// OptionalCyclic Plc -> Rob
AxesGroup.Config.PlcToRob.Header.TelegramNumberPlcToRob.00 := AxesGroup.Parameter.OptionalCyclic.PlcToRob.UseCallSubprogram;
AxesGroup.Config.PlcToRob.Header.TelegramNumberPlcToRob.01 := AxesGroup.Parameter.OptionalCyclic.PlcToRob.UseCartesianPos;
AxesGroup.Config.PlcToRob.Header.TelegramNumberPlcToRob.02 := AxesGroup.Parameter.OptionalCyclic.PlcToRob.UseJointPos;
AxesGroup.Config.PlcToRob.Header.TelegramNumberPlcToRob.03 := AxesGroup.Parameter.OptionalCyclic.PlcToRob.UseForce;
AxesGroup.Config.PlcToRob.Header.TelegramNumberPlcToRob.04 := AxesGroup.Parameter.OptionalCyclic.PlcToRob.Bit04;
AxesGroup.Config.PlcToRob.Header.TelegramNumberPlcToRob.05 := AxesGroup.Parameter.OptionalCyclic.PlcToRob.Bit05;
AxesGroup.Config.PlcToRob.Header.TelegramNumberPlcToRob.06 := AxesGroup.Parameter.OptionalCyclic.PlcToRob.Bit06;
AxesGroup.Config.PlcToRob.Header.TelegramNumberPlcToRob.07 := AxesGroup.Parameter.OptionalCyclic.PlcToRob.Bit07;  
AxesGroup.Config.PlcToRob.Header.TelegramNumberPlcToRob.08 := AxesGroup.Parameter.OptionalCyclic.PlcToRob.UseTwoSequences;
AxesGroup.Config.PlcToRob.Header.TelegramNumberPlcToRob.09 := AxesGroup.Parameter.OptionalCyclic.PlcToRob.UseCartesianPositionExt;
AxesGroup.Config.PlcToRob.Header.TelegramNumberPlcToRob.10 := AxesGroup.Parameter.OptionalCyclic.PlcToRob.UseJointPositionExt;
AxesGroup.Config.PlcToRob.Header.TelegramNumberPlcToRob.11 := AxesGroup.Parameter.OptionalCyclic.PlcToRob.Bit11;
AxesGroup.Config.PlcToRob.Header.TelegramNumberPlcToRob.12 := AxesGroup.Parameter.OptionalCyclic.PlcToRob.Bit12;
AxesGroup.Config.PlcToRob.Header.TelegramNumberPlcToRob.13 := AxesGroup.Parameter.OptionalCyclic.PlcToRob.Bit13;
AxesGroup.Config.PlcToRob.Header.TelegramNumberPlcToRob.14 := AxesGroup.Parameter.OptionalCyclic.PlcToRob.Bit14;
AxesGroup.Config.PlcToRob.Header.TelegramNumberPlcToRob.15 := AxesGroup.Parameter.OptionalCyclic.PlcToRob.Bit15;  

// OptionalCyclic Rob -> Plc
AxesGroup.Config.PlcToRob.Header.TelegramNumberPlcToRob.00 := AxesGroup.Parameter.OptionalCyclic.RobToPlc.UseCallSubprogram;
AxesGroup.Config.PlcToRob.Header.TelegramNumberPlcToRob.01 := AxesGroup.Parameter.OptionalCyclic.RobToPlc.UseCartesianPos;
AxesGroup.Config.PlcToRob.Header.TelegramNumberPlcToRob.02 := AxesGroup.Parameter.OptionalCyclic.RobToPlc.UseJointPos;
AxesGroup.Config.PlcToRob.Header.TelegramNumberPlcToRob.03 := AxesGroup.Parameter.OptionalCyclic.RobToPlc.UseForce;
AxesGroup.Config.PlcToRob.Header.TelegramNumberPlcToRob.04 := AxesGroup.Parameter.OptionalCyclic.RobToPlc.UseCurrent;
AxesGroup.Config.PlcToRob.Header.TelegramNumberPlcToRob.05 := AxesGroup.Parameter.OptionalCyclic.RobToPlc.Bit05;
AxesGroup.Config.PlcToRob.Header.TelegramNumberPlcToRob.06 := AxesGroup.Parameter.OptionalCyclic.RobToPlc.Bit06;
AxesGroup.Config.PlcToRob.Header.TelegramNumberPlcToRob.07 := AxesGroup.Parameter.OptionalCyclic.RobToPlc.Bit07;  
AxesGroup.Config.PlcToRob.Header.TelegramNumberPlcToRob.08 := AxesGroup.Parameter.OptionalCyclic.RobToPlc.UseTwoSequences;
AxesGroup.Config.PlcToRob.Header.TelegramNumberPlcToRob.09 := AxesGroup.Parameter.OptionalCyclic.RobToPlc.UseCartesianPositionExt;
AxesGroup.Config.PlcToRob.Header.TelegramNumberPlcToRob.10 := AxesGroup.Parameter.OptionalCyclic.RobToPlc.UseJointPositionExt;
AxesGroup.Config.PlcToRob.Header.TelegramNumberPlcToRob.11 := AxesGroup.Parameter.OptionalCyclic.RobToPlc.UseForceExt;
AxesGroup.Config.PlcToRob.Header.TelegramNumberPlcToRob.12 := AxesGroup.Parameter.OptionalCyclic.RobToPlc.UseCurrentEct;
AxesGroup.Config.PlcToRob.Header.TelegramNumberPlcToRob.13 := AxesGroup.Parameter.OptionalCyclic.RobToPlc.Bit13;  
AxesGroup.Config.PlcToRob.Header.TelegramNumberPlcToRob.14 := AxesGroup.Parameter.OptionalCyclic.RobToPlc.Bit14;
AxesGroup.Config.PlcToRob.Header.TelegramNumberPlcToRob.15 := AxesGroup.Parameter.OptionalCyclic.RobToPlc.Bit15;  


AxesGroup.Config.PlcToRob.Header.ClientDate := DATE_TO_IEC_DATE(DATE#2024-06-01 ); {warning 'ToDo: Get current date from target system'}
AxesGroup.Config.PlcToRob.Header.ClientTime := TIME_TO_IEC_TIME(TOD#12:00:00.000); {warning 'ToDo: Get current time from target system'}

// reset all variables
SendData.Reset();

// PlcToRob.Cyclic {{{
  
// PlcToRob.Cyclic.SRCIVersion  
SendData.AddByte     (VersionToByte(AxesGroup.Config.PlcToRob.Header.SRCIVersion));
// PlcToRob.Cyclic.FastStop_LifeSign
SendData.AddHalfBytes(AxesGroup.Config.PlcToRob.Header.FastStop, AxesGroup.Config.PlcToRob.Header.LifeSign); 
// PlcToRob.Cyclic.TelegramLengthPlcToRob
SendData.AddUint     (AxesGroup.Config.PlcToRob.Header.TelegramLengthPlcToRob);
// PlcToRob.Cyclic.TelegramLengthRobToPlc 
SendData.AddUint     (AxesGroup.Config.PlcToRob.Header.TelegramLengthRobToPlc);
// PlcToRob.Cyclic.AxesGroupID_Control
SendData.AddHalfBytes(AxesGroup.Config.PlcToRob.Header.AxesGroupID, AxesGroup.Config.PlcToRob.Header.Control);
// PlcToRob.Cyclic.Reserved
SendData.AddByte     (AxesGroup.Config.PlcToRob.Header.Reserved);
// PlcToRob.Cyclic.TelegramNumberPlcToRob 
SendData.AddUint     (AxesGroup.Config.PlcToRob.Header.TelegramNumberPlcToRob);
// PlcToRob.Cyclic.TelegramNumberRobToPlc 
SendData.AddUint     (AxesGroup.Config.PlcToRob.Header.TelegramNumberRobToPlc);
// PlcToRob.Cyclic.ClientDate
SendData.AddUint     (AxesGroup.Config.PlcToRob.Header.ClientDate); 
// PlcToRob.Cyclic.ClientTime
SendData.AddTime     (AxesGroup.Config.PlcToRob.Header.ClientTime);  
// }}}

// PlcToRob.CyclicOptional Data {{{

// AxesGroup.OptionalCyclic.PlcToRob.SubProgramData {{{
IF ( AxesGroup.OptionalCyclic.PlcToRob.SubProgramData.Active )
THEN
  SendData.AddDataBlock( ADR(AxesGroup.OptionalCyclic.PlcToRob.SubProgramData.Data), SIZEOF(AxesGroup.OptionalCyclic.PlcToRob.SubProgramData.Data));  
END_IF
// }}}

// AxesGroup.OptionalCyclic.PlcToRob.CartesianPos {{{
IF ( AxesGroup.OptionalCyclic.PlcToRob.CartesianPosition.Active) 
THEN
  // AxesGroup.OptionalCyclic.PlcToRob.CartesianPos.X
  SendData.AddReal(AxesGroup.OptionalCyclic.PlcToRob.CartesianPosition.X);
  // AxesGroup.OptionalCyclic.PlcToRob.CartesianPos.Y
  SendData.AddReal( AxesGroup.OptionalCyclic.PlcToRob.CartesianPosition.Y);
  // AxesGroup.OptionalCyclic.PlcToRob.CartesianPos.Z
  SendData.AddReal( AxesGroup.OptionalCyclic.PlcToRob.CartesianPosition.Z);
  // AxesGroup.OptionalCyclic.PlcToRob.CartesianPos.Rx
  SendData.AddReal( AxesGroup.OptionalCyclic.PlcToRob.CartesianPosition.Rx);
  // AxesGroup.OptionalCyclic.PlcToRob.CartesianPos.Ry
  SendData.AddReal( AxesGroup.OptionalCyclic.PlcToRob.CartesianPosition.Ry);
  // AxesGroup.OptionalCyclic.PlcToRob.CartesianPos.Rz
  SendData.AddReal( AxesGroup.OptionalCyclic.PlcToRob.CartesianPosition.Rz);
  // AxesGroup.OptionalCyclic.PlcToRob.CartesianPos.Config
 _tmpByte   := 0;
 _tmpByte.0 := AxesGroup.OptionalCyclic.PlcToRob.CartesianPosition.Config.Shoulder = ArmConfigShoulder.BACK;
 _tmpByte.1 := AxesGroup.OptionalCyclic.PlcToRob.CartesianPosition.Config.Elbow    = ArmConfigElbow   .DOWN;
 _tmpByte.2 := AxesGroup.OptionalCyclic.PlcToRob.CartesianPosition.Config.Wrist    = ArmConfigWrist   .FLIP;
 
  SendData.AddByte(_tmpByte);
          
  // AxesGroup.OptionalCyclic.PlcToRob.CartesianPos.TurnNumber.J1 + J2
  SendData.AddHalfBytes( SINT_TO_BYTE(AxesGroup.OptionalCyclic.PlcToRob.CartesianPosition.TurnNumber.J1Turns), SINT_TO_BYTE(AxesGroup.OptionalCyclic.PlcToRob.CartesianPosition.TurnNumber.J2Turns));
  // AxesGroup.OptionalCyclic.PlcToRob.CartesianPos.TurnNumber.J3 + J4
  SendData.AddHalfBytes( SINT_TO_BYTE(AxesGroup.OptionalCyclic.PlcToRob.CartesianPosition.TurnNumber.J3Turns), SINT_TO_BYTE(AxesGroup.OptionalCyclic.PlcToRob.CartesianPosition.TurnNumber.J4Turns));
  // AxesGroup.OptionalCyclic.PlcToRob.CartesianPos.TurnNumber.J5 + J6
  SendData.AddHalfBytes( SINT_TO_BYTE(AxesGroup.OptionalCyclic.PlcToRob.CartesianPosition.TurnNumber.J5Turns), SINT_TO_BYTE(AxesGroup.OptionalCyclic.PlcToRob.CartesianPosition.TurnNumber.J6Turns));
  // AxesGroup.OptionalCyclic.PlcToRob.CartesianPos.TurnNumber.E1 
  SendData.AddSint(AxesGroup.OptionalCyclic.PlcToRob.CartesianPosition.TurnNumber.E1Turns);
  // AxesGroup.OptionalCyclic.PlcToRob.CartesianPos.E1
  SendData.AddReal( AxesGroup.OptionalCyclic.PlcToRob.CartesianPosition.E1);
  // AxesGroup.OptionalCyclic.PlcToRob.CartesianPos.CoordinateSystem.ToolNo
  SendData.AddUsint(AxesGroup.OptionalCyclic.PlcToRob.CartesianPosition.CoordinateSystem.ToolNo);
  // AxesGroup.OptionalCyclic.PlcToRob.CartesianPos.CoordinateSystem.FrameNo 
  SendData.AddUsint(AxesGroup.OptionalCyclic.PlcToRob.CartesianPosition.CoordinateSystem.FrameNo);  
END_IF
// }}}
  
// AxesGroup.OptionalCyclic.PlcToRob.CartesianPosExt {{{
IF ( AxesGroup.OptionalCyclic.PlcToRob.CartesianPositionExt.Active) 
THEN
  // AxesGroup.OptionalCyclic.PlcToRob.CartesianPosExt.E2 
  SendData.AddReal( AxesGroup.OptionalCyclic.PlcToRob.CartesianPositionExt.E2);
  // AxesGroup.OptionalCyclic.PlcToRob.CartesianPosExt.E3
  SendData.AddReal( AxesGroup.OptionalCyclic.PlcToRob.CartesianPositionExt.E3);
  // AxesGroup.OptionalCyclic.PlcToRob.CartesianPosExt.E4
  SendData.AddReal( AxesGroup.OptionalCyclic.PlcToRob.CartesianPositionExt.E4);
  // AxesGroup.OptionalCyclic.PlcToRob.CartesianPosExt.E5
  SendData.AddReal( AxesGroup.OptionalCyclic.PlcToRob.CartesianPositionExt.E5);
  // AxesGroup.OptionalCyclic.PlcToRob.CartesianPosExt.E6
  SendData.AddReal( AxesGroup.OptionalCyclic.PlcToRob.CartesianPositionExt.E6);
END_IF    
// }}}
      
// AxesGroup.OptionalCyclic.PlcToRob.JointPosition {{{
IF ( AxesGroup.OptionalCyclic.PlcToRob.JointPosition.Active) 
THEN
  // AxesGroup.OptionalCyclic.PlcToRob.JointPosition.J1
  SendData.AddReal( AxesGroup.OptionalCyclic.PlcToRob.JointPosition.J1);
  // AxesGroup.OptionalCyclic.PlcToRob.JointPosition.J2
  SendData.AddReal( AxesGroup.OptionalCyclic.PlcToRob.JointPosition.J2);
  // AxesGroup.OptionalCyclic.PlcToRob.JointPosition.J3
  SendData.AddReal( AxesGroup.OptionalCyclic.PlcToRob.JointPosition.J3);
  // AxesGroup.OptionalCyclic.PlcToRob.JointPosition.J4
  SendData.AddReal( AxesGroup.OptionalCyclic.PlcToRob.JointPosition.J4);
  // AxesGroup.OptionalCyclic.PlcToRob.JointPosition.J5
  SendData.AddReal( AxesGroup.OptionalCyclic.PlcToRob.JointPosition.J5);
  // AxesGroup.OptionalCyclic.PlcToRob.JointPosition.J6
  SendData.AddReal( AxesGroup.OptionalCyclic.PlcToRob.JointPosition.J6);
  // AxesGroup.OptionalCyclic.PlcToRob.JointPosition.E1
  SendData.AddReal( AxesGroup.OptionalCyclic.PlcToRob.JointPosition.E1);
END_IF
// }}}

// AxesGroup.OptionalCyclic.PlcToRob.JointPositionExt {{{
IF ( AxesGroup.OptionalCyclic.PlcToRob.JointPositionExt.Active) 
THEN
  // AxesGroup.OptionalCyclic.PlcToRob.JointPositionExt.E2
  SendData.AddReal( AxesGroup.OptionalCyclic.PlcToRob.JointPositionExt.E2);
  // AxesGroup.OptionalCyclic.PlcToRob.JointPositionExt.E3
  SendData.AddReal( AxesGroup.OptionalCyclic.PlcToRob.JointPositionExt.E3);  
  // AxesGroup.OptionalCyclic.PlcToRob.JointPositionExt.E4
  SendData.AddReal( AxesGroup.OptionalCyclic.PlcToRob.JointPositionExt.E4);
  // AxesGroup.OptionalCyclic.PlcToRob.JointPositionExt.E5
  SendData.AddReal( AxesGroup.OptionalCyclic.PlcToRob.JointPositionExt.E5);
  // AxesGroup.OptionalCyclic.PlcToRob.JointPositionExt.E6
  SendData.AddReal( AxesGroup.OptionalCyclic.PlcToRob.JointPositionExt.E6);        
END_IF  
// }}}
     
// AxesGroup.OptionalCyclic.PlcToRob.CartesianForce {{{
IF ( AxesGroup.OptionalCyclic.PlcToRob.CartesianForce.Active) 
THEN
  // AxesGroup.OptionalCyclic.PlcToRob.CartesianForce.X
  SendData.AddReal( AxesGroup.OptionalCyclic.PlcToRob.CartesianForce.X);
  // AxesGroup.OptionalCyclic.PlcToRob.CartesianForce.Y
  SendData.AddReal( AxesGroup.OptionalCyclic.PlcToRob.CartesianForce.Y);
  // AxesGroup.OptionalCyclic.PlcToRob.CartesianForce.Z
  SendData.AddReal( AxesGroup.OptionalCyclic.PlcToRob.CartesianForce.Z);
  // AxesGroup.OptionalCyclic.PlcToRob.CartesianForce.Rx
  SendData.AddReal( AxesGroup.OptionalCyclic.PlcToRob.CartesianForce.Rx);
  // AxesGroup.OptionalCyclic.PlcToRob.CartesianForce.Ry
  SendData.AddReal( AxesGroup.OptionalCyclic.PlcToRob.CartesianForce.Ry);
  // AxesGroup.OptionalCyclic.PlcToRob.CartesianForce.Rz
  SendData.AddReal( AxesGroup.OptionalCyclic.PlcToRob.CartesianForce.Rz);
END_IF  
// }}}
                    
// AxesGroup.OptionalCyclic.PlcToRob.CartesianForceExt {{{
IF ( AxesGroup.OptionalCyclic.PlcToRob.CartesianForceExt.Active) 
THEN
  // AxesGroup.OptionalCyclic.PlcToRob.CartesianForceExt.E1
  SendData.AddReal( AxesGroup.OptionalCyclic.PlcToRob.CartesianForceExt.E1);
  // AxesGroup.OptionalCyclic.PlcToRob.CartesianForceExt.E2
  SendData.AddReal( AxesGroup.OptionalCyclic.PlcToRob.CartesianForceExt.E2);
  // AxesGroup.OptionalCyclic.PlcToRob.CartesianForceExt.E3
  SendData.AddReal( AxesGroup.OptionalCyclic.PlcToRob.CartesianForceExt.E3);
  // AxesGroup.OptionalCyclic.PlcToRob.CartesianForceExt.E4
  SendData.AddReal( AxesGroup.OptionalCyclic.PlcToRob.CartesianForceExt.E4);
  // AxesGroup.OptionalCyclic.PlcToRob.CartesianForceExt.E5
  SendData.AddReal( AxesGroup.OptionalCyclic.PlcToRob.CartesianForceExt.E5);
  // AxesGroup.OptionalCyclic.PlcToRob.CartesianForceExt.E6
  SendData.AddReal( AxesGroup.OptionalCyclic.PlcToRob.CartesianForceExt.E6);
END_IF                    


// }}}

// }}}
  
{warning 'ToDo: Sequence Handling for Seq 0..1'}
// PlcToRob.Sequence[0]{{{

// PlcToRob.Sequence[0].Header{{{
  
// AxesGroup.OptionalCyclic.PlcToRob.Sequence[0].Header.SEQ_ACK 
SendData.AddUint( Telegram.PlcToRob.Sequence[0].Header.SEQ_ACK);
// AxesGroup.OptionalCyclic.PlcToRob.Sequence[0].Header.PayloadLength
SendData.AddUint( Telegram.PlcToRob.Sequence[0].Header.PayloadLength);
// }}}

    
{warning 'ToDo: Fragment Handling for Frag 0..9'}
// PlcToRob.Sequence[0].Fragment {{{

       
          
// PlcToRob.Sequence[0].Fragment.Header {{{

// AxesGroup.OptionalCyclic.PlcToRob.Sequence[0].Fragment.Header.ID 
SendData.AddUint( Telegram.PlcToRob.Sequence[0].Fragment[0].Header.ID);
// AxesGroup.OptionalCyclic.PlcToRob.Sequence[0].Fragment.Header.Reserve
SendData.AddByte(Telegram.PlcToRob.Sequence[0].Fragment[0].Header.Reserve);
// AxesGroup.OptionalCyclic.PlcToRob.Sequence[0].Fragment.Header.FragmentAction 
SendData.AddByte(FragmentActionToByte(Telegram.PlcToRob.Sequence[0].Fragment[0].Header.FragmentAction));
// AxesGroup.OptionalCyclic.PlcToRob.Sequence[0].Fragment.Header.PayloadPointer
SendData.AddUint(Telegram.PlcToRob.Sequence[0].Fragment[0].Header.PayloadPointer);
// AxesGroup.OptionalCyclic.PlcToRob.Sequence[0].Fragment.Header.PayloadLength 
SendData.AddUint(Telegram.PlcToRob.Sequence[0].Fragment[0].Header.PayloadLength);

// PlcToRob.Sequence[0].Fragment.Command {{{    
FOR _payLoadPtr := AxesGroup.Acyclic.ActiveCommandRegister.Register[1].Command[1].PayLoadPtr TO AxesGroup.Acyclic.ActiveCommandRegister.Register[1].Command[1].PayloadLen   
DO
  // copy payload
  SendData.AddByte(AxesGroup.Acyclic.ActiveCommandRegister.Register[1].Command[1].Payload[_payLoadPtr]);

  // inc payload pointer
  AxesGroup.Acyclic.ActiveCommandRegister.Register[1].Command[1].PayLoadPtr 
    := AxesGroup.Acyclic.ActiveCommandRegister.Register[1].Command[1].PayLoadPtr + 1;

  // set command state
  IF ( AxesGroup.Acyclic.ActiveCommandRegister.Register[1].Command[1].PayLoadPtr >= AxesGroup.Acyclic.ActiveCommandRegister.Register[1].Command[1].PayLoadLen) 
  THEN
    AxesGroup.Acyclic.ActiveCommandRegister.Register[1].Command[1].State := BufferStateCmd.PROCESSED;
  ELSE
    AxesGroup.Acyclic.ActiveCommandRegister.Register[1].Command[1].State := BufferStateCmd.SENDING;  
  END_IF 

  // check limit reached ?
  IF ( SendData.PayloadLen >= RobotLibraryParameter.ROBOT_OUT_DATA_MAX - SIZEOF(Telegram.PlcToRob.Footer)) 
  THEN
    EXIT;
  END_IF  
END_FOR    
// }}}
// }}}
// }}}
// }}}


// Footer {{{

// PlcToRob.Footer.Reserved_LifeSign
SendData.AddHalfBytes(0, AxesGroup.Config.PlcToRob.Header.LifeSign);

// }}}

                      
END_METHOD

METHOD NetworkLayer
VAR_IN_OUT
  /// Robot assignment of function
  AxesGroup         : AxesGroup;
    /// Inputs of PLC for communication from RC
  RobotInData       : ARRAY[1..RobotLibraryParameter.ROBOT_IN_DATA_MAX ] OF BYTE;
  /// Outputs of PLC for communication to RC
  RobotOutData      : ARRAY[1..RobotLibraryParameter.ROBOT_OUT_DATA_MAX] OF BYTE;
END_VAR
                        CreateSendData   ( AxesGroup    := AxesGroup,
                   RobotInData  := RobotInData,
                   RobotOutData := RobotOutData );

ParseRecvData    ( AxesGroup    := AxesGroup,
                   RobotInData  := RobotInData,
                   RobotOutData := RobotOutData );                   
                      
END_METHOD

METHOD OnCall
VAR_IN_OUT
   /// Robot assignment of function
  AxesGroup : AxesGroup;
END_VAR
                        
                      
END_METHOD

METHOD ParseRecvData
VAR_IN_OUT
  /// Robot assignment of function
  AxesGroup    : AxesGroup;
  /// Inputs of PLC for communication from RC
  RobotInData  : ARRAY[1..RobotLibraryParameter.ROBOT_IN_DATA_MAX ] OF BYTE;
  /// Outputs of PLC for communication to RC
  RobotOutData : ARRAY[1..RobotLibraryParameter.ROBOT_OUT_DATA_MAX] OF BYTE;
END_VAR

VAR
  /// internal index
 _idx             : DINT;
  /// temporary DWORD
 _tmpDword        : DWORD;
  /// length of data block
 _dataBlockLength : UINT;
  /// internal payload length
 _payLoadLen      : DWORD;  
  /// internal payload pointer
 _payLoadPtr      : DWORD;  
END_VAR
                        // Version
AxesGroup.Config.RobToPlc.Header.SRCIVersion.MajorVersion := RecvData.GetUsint();
AxesGroup.Config.RobToPlc.Header.SRCIVersion.MinorVersion := RecvData.GetUsint();
AxesGroup.Config.RobToPlc.Header.SRCIVersion.PatchVersion := RecvData.GetUsint();
// Connection alive signal
AxesGroup.Config.RobToPlc.Header.LifeSign       := RecvData.GetByte();
// Reserved byte
AxesGroup.Config.RobToPlc.Header.Reserved       := RecvData.GetByte();
// Initialization and Telegram control state
AxesGroup.Config.RobToPlc.Header.TelegramState  := RecvData.GetUsint();
// Combination of various RA related states.
AxesGroup.Config.RobToPlc.Header.StatusRobotArm := DwordToRaStatusWord(RecvData.GetDword());
// Actual override in percentage encoding 
AxesGroup.Config.RobToPlc.Header.Override       := RecvData.GetUint();


// AxesGroup.OptionalCyclic {{{

// AxesGroup.OptionalCyclic.RobToPlc.SubProgramData {{{
IF ( AxesGroup.OptionalCyclic.RobToPlc.SubProgramData.Active )
THEN
  FOR _idx := 0 TO 25 DO
    AxesGroup.Config.RobToPlc.CyclicOptional.SubProgramData.Data[_idx] := RecvData.GetByte(); 
	END_FOR
END_IF
// }}}
  
// AxesGroup.OptionalCyclic.RobToPlc.CartesianPos {{{
IF ( AxesGroup.OptionalCyclic.RobToPlc.CartesianPosition.Active )
THEN
  AxesGroup.Config.RobToPlc.CyclicOptional.CartesianPosition.X                    := RecvData.GetReal();
  AxesGroup.Config.RobToPlc.CyclicOptional.CartesianPosition.Y                    := RecvData.GetReal();
  AxesGroup.Config.RobToPlc.CyclicOptional.CartesianPosition.Z                    := RecvData.GetReal();
  AxesGroup.Config.RobToPlc.CyclicOptional.CartesianPosition.Rx                   := RecvData.GetReal();
  AxesGroup.Config.RobToPlc.CyclicOptional.CartesianPosition.Ry                   := RecvData.GetReal();
  AxesGroup.Config.RobToPlc.CyclicOptional.CartesianPosition.Rz                   := RecvData.GetReal();
  AxesGroup.Config.RobToPlc.CyclicOptional.CartesianPosition.Config               := RecvData.GetArmConfig();
  AxesGroup.Config.RobToPlc.CyclicOptional.CartesianPosition.TurnNumber           := RecvData.GetTurnNumbers();
  AxesGroup.Config.RobToPlc.CyclicOptional.CartesianPosition.E1                   := RecvData.GetReal();  
  AxesGroup.Config.RobToPlc.CyclicOptional.CartesianPosition.E2                   := RecvData.GetReal();
  AxesGroup.Config.RobToPlc.CyclicOptional.CartesianPosition.E3                   := RecvData.GetReal();
  AxesGroup.Config.RobToPlc.CyclicOptional.CartesianPosition.E4                   := RecvData.GetReal();
  AxesGroup.Config.RobToPlc.CyclicOptional.CartesianPosition.E5                   := RecvData.GetReal();
  AxesGroup.Config.RobToPlc.CyclicOptional.CartesianPosition.E6                   := RecvData.GetReal();      
  AxesGroup.Config.RobToPlc.CyclicOptional.CartesianPosition.ToolNo               := RecvData.GetUsint();
  AxesGroup.Config.RobToPlc.CyclicOptional.CartesianPosition.FrameNo              := RecvData.GetUsint();
  AxesGroup.Config.RobToPlc.CyclicOptional.CartesianPosition.CurrentlyUsedToolNo  := RecvData.GetUsint();
  AxesGroup.Config.RobToPlc.CyclicOptional.CartesianPosition.CurrentlyUsedFrameNo := RecvData.GetUsint();
  AxesGroup.Config.RobToPlc.CyclicOptional.CartesianPosition.Reserve_1            := RecvData.GetByte();
  AxesGroup.Config.RobToPlc.CyclicOptional.CartesianPosition.Reserve_2            := RecvData.GetByte();  
END_IF
// }}}

// AxesGroup.OptionalCyclic.RobToPlc.CartesianPosExt {{{
IF ( AxesGroup.OptionalCyclic.RobToPlc.CartesianPositionExt.Active )
THEN
  AxesGroup.Config.RobToPlc.CyclicOptional.CartesianPositionExt.E2 := RecvData.GetReal();
  AxesGroup.Config.RobToPlc.CyclicOptional.CartesianPositionExt.E3 := RecvData.GetReal();
  AxesGroup.Config.RobToPlc.CyclicOptional.CartesianPositionExt.E4 := RecvData.GetReal();
  AxesGroup.Config.RobToPlc.CyclicOptional.CartesianPositionExt.E5 := RecvData.GetReal();
  AxesGroup.Config.RobToPlc.CyclicOptional.CartesianPositionExt.E6 := RecvData.GetReal();
END_IF  
// }}}       

// AxesGroup.OptionalCyclic.RobToPlc.JointPosition {{{
IF ( AxesGroup.OptionalCyclic.RobToPlc.JointPosition.Active )
THEN
  AxesGroup.Config.RobToPlc.CyclicOptional.JointPosition.J1         := RecvData.GetReal();
  AxesGroup.Config.RobToPlc.CyclicOptional.JointPosition.J2         := RecvData.GetReal();
  AxesGroup.Config.RobToPlc.CyclicOptional.JointPosition.J3         := RecvData.GetReal();
  AxesGroup.Config.RobToPlc.CyclicOptional.JointPosition.J4         := RecvData.GetReal();
  AxesGroup.Config.RobToPlc.CyclicOptional.JointPosition.J5         := RecvData.GetReal();
  AxesGroup.Config.RobToPlc.CyclicOptional.JointPosition.J6         := RecvData.GetReal();
  AxesGroup.Config.RobToPlc.CyclicOptional.JointPosition.E1         := RecvData.GetReal();
  AxesGroup.Config.RobToPlc.CyclicOptional.JointPosition.E1_Reserve := RecvData.GetWord();
END_IF  
// }}}
  
// AxesGroup.OptionalCyclic.RobToPlc.JointPosition {{{
IF ( AxesGroup.OptionalCyclic.RobToPlc.JointPositionExt.Active )
THEN
  AxesGroup.Config.RobToPlc.CyclicOptional.JointPositionExt.E2 := RecvData.GetReal();
  AxesGroup.Config.RobToPlc.CyclicOptional.JointPositionExt.E3 := RecvData.GetReal();
  AxesGroup.Config.RobToPlc.CyclicOptional.JointPositionExt.E4 := RecvData.GetReal();
  AxesGroup.Config.RobToPlc.CyclicOptional.JointPositionExt.E5 := RecvData.GetReal();
  AxesGroup.Config.RobToPlc.CyclicOptional.JointPositionExt.E6 := RecvData.GetReal();  
END_IF  
// }}}    
      
// AxesGroup.OptionalCyclic.RobToPlc.CartesianForce {{{
IF ( AxesGroup.OptionalCyclic.RobToPlc.CartesianForce.Active )
THEN
  AxesGroup.Config.RobToPlc.CyclicOptional.Force.X  := RecvData.GetReal();
  AxesGroup.Config.RobToPlc.CyclicOptional.Force.Y  := RecvData.GetReal();
  AxesGroup.Config.RobToPlc.CyclicOptional.Force.Z  := RecvData.GetReal();
  AxesGroup.Config.RobToPlc.CyclicOptional.Force.Rx := RecvData.GetReal();
  AxesGroup.Config.RobToPlc.CyclicOptional.Force.Ry := RecvData.GetReal();
  AxesGroup.Config.RobToPlc.CyclicOptional.Force.Rz := RecvData.GetReal();
END_IF  
// }}}    
      
// AxesGroup.OptionalCyclic.RobToPlc.CartesianForceExt {{{
IF ( AxesGroup.OptionalCyclic.RobToPlc.CartesianForceExt.Active )
THEN
  AxesGroup.Config.RobToPlc.CyclicOptional.ForceExt.E1  := RecvData.GetReal();
  AxesGroup.Config.RobToPlc.CyclicOptional.ForceExt.E2  := RecvData.GetReal();
  AxesGroup.Config.RobToPlc.CyclicOptional.ForceExt.E3  := RecvData.GetReal();
  AxesGroup.Config.RobToPlc.CyclicOptional.ForceExt.E4  := RecvData.GetReal();
  AxesGroup.Config.RobToPlc.CyclicOptional.ForceExt.E5  := RecvData.GetReal();
  AxesGroup.Config.RobToPlc.CyclicOptional.ForceExt.E6  := RecvData.GetReal();
END_IF
// }}}    

// AxesGroup.OptionalCyclic.RobToPlc.Current {{{
IF ( AxesGroup.OptionalCyclic.RobToPlc.JointCurrent.Active )
THEN
  AxesGroup.Config.RobToPlc.CyclicOptional.Current.J1  := RecvData.GetReal();
  AxesGroup.Config.RobToPlc.CyclicOptional.Current.J2  := RecvData.GetReal();
  AxesGroup.Config.RobToPlc.CyclicOptional.Current.J3  := RecvData.GetReal();
  AxesGroup.Config.RobToPlc.CyclicOptional.Current.J4  := RecvData.GetReal();
  AxesGroup.Config.RobToPlc.CyclicOptional.Current.J5  := RecvData.GetReal();
  AxesGroup.Config.RobToPlc.CyclicOptional.Current.J6  := RecvData.GetReal();
END_IF
// }}}    
  
// AxesGroup.OptionalCyclic.RobToPlc.CurrentExt {{{
IF ( AxesGroup.OptionalCyclic.RobToPlc.JointCurrentExt.Active )
THEN
  AxesGroup.Config.RobToPlc.CyclicOptional.CurrentExt.E1  := RecvData.GetReal();
  AxesGroup.Config.RobToPlc.CyclicOptional.CurrentExt.E2  := RecvData.GetReal();
  AxesGroup.Config.RobToPlc.CyclicOptional.CurrentExt.E3  := RecvData.GetReal();
  AxesGroup.Config.RobToPlc.CyclicOptional.CurrentExt.E4  := RecvData.GetReal();
  AxesGroup.Config.RobToPlc.CyclicOptional.CurrentExt.E5  := RecvData.GetReal();
  AxesGroup.Config.RobToPlc.CyclicOptional.CurrentExt.E6  := RecvData.GetReal();
END_IF
// }}}
    
// }}}    

// Sequence Data
AxesGroup.Config.RobToPlc.Sequence[0].Header.SEQ_ACK       := RecvData.GetUint();
AxesGroup.Config.RobToPlc.Sequence[0].Header.PayloadLength := RecvData.GetUint();

AxesGroup.Config.RobToPlc.Sequence[0].Fragment[1].Header.ID                  := RecvData.GetUint();
AxesGroup.Config.RobToPlc.Sequence[0].Fragment[1].Header.Reserve             := RecvData.GetByte();
AxesGroup.Config.RobToPlc.Sequence[0].Fragment[1].Header.FragmentAction      := RecvData.GetFragmentAction();
AxesGroup.Config.RobToPlc.Sequence[0].Fragment[1].Header.PayloadPointer      := RecvData.GetUint();
AxesGroup.Config.RobToPlc.Sequence[0].Fragment[1].Header.PayloadLength       := RecvData.GetUint();

AxesGroup.Config.RobToPlc.Sequence[0].Fragment[1].Command.Header.CmdType     := RecvData.GetUint();
AxesGroup.Config.RobToPlc.Sequence[0].Fragment[1].Command.Header.Prio        := RecvData.GetByte();
AxesGroup.Config.RobToPlc.Sequence[0].Fragment[1].Command.Header.ExecMode    := RecvData.GetUsint();
AxesGroup.Config.RobToPlc.Sequence[0].Fragment[1].Command.Header.ParSequence := RecvData.GetByte();


_dataBlockLength :=           AxesGroup.Config.RobToPlc.Sequence[0].Fragment[1].Header.PayloadLength 
                    -  SIZEOF(AxesGroup.Config.RobToPlc.Sequence[0].Fragment[1].Command.Header); 

FOR _idx := 1 TO  _dataBlockLength
DO
  AxesGroup.Config.RobToPlc.Sequence[0].Fragment[1].Command.Payload[_idx] := RecvData.GetByte();
END_FOR

WHILE (RecvData.PayloadPtr < 1)
DO
;  
END_WHILE
                      
END_METHOD

METHOD TransportLayer
VAR_IN_OUT
   /// Robot assignment of function
  AxesGroup : AxesGroup;
END_VAR
                        
                      
END_METHOD
END_FUNCTION_BLOCK

/// Calculate frame with three-point method
FUNCTION_BLOCK CalculateFrameFB EXTENDS RobotLibraryBaseFB
// ------------------------------------------------------------------------- 
//  SRCI Robot Library                                                
// ------------------------------------------------------------------------- 
//                                                                           
//  Object:      CalculateFrameFB                                       
//  Author:      Thorsten Brach                                                
//  Date:        2024-06-01
//
//  Description:                                              
//   
//                                                                           
//  Copyright: 
//    (C) 2024 Thorsten Brach. All rights reserved                                                                         
//                                                                           
//  Disclaimer:                                                                           
//    This project is provided without any guarantee and can be used for   
//    private and commercial purposes. Any commercial use is at the user’s 
//    own risk and responsibility.
//
// -------------------------------------------------------------------------
VAR_INPUT
  /// Start of the command at the rising edge
  Execute            : BOOL;
  /// Define which method should be used to calculate the tool frame
  Mode               : FrameCalculationMode;
  /// Index of target frame
  /// • 0: WCS (default)
  /// • 1..254: User frames
  FrameNo            : USINT;  
  /// Cartesian position in the positive direction of the  X-Axis of the calculated frame coordinate system relative to the given frame
  Position_X         : RobotCartesianPosition;
  /// Cartesian position in the XY-plane of the calculated frame coordinate system relative to the given frame.
  Position_XY        : RobotCartesianPosition;
  /// Cartesian position of the origin of the calculated frame coordinate system relative to the given frame.
  Position_Origin    : RobotCartesianPosition;
  /// Cartesian position of the postponement of the origin of the calculated frame coordinate system relative to the given frame.
  /// Auxiliary position if the origin of the can’t be reached by the robot, i.e. because it is inside an object.
  OriginShift        : RobotCartesianPosition;
  /// Index of frame on which the calculated frame is depending
  /// •      0: WCS (default)
  /// • 1..254: User frames
  ReferenceFrame     : USINT;
END_VAR
VAR_OUTPUT
  /// The command has been completed successfully
  Done               : BOOL;
  /// FB is being processed
  Busy               : BOOL;
  /// Command is transferred and confirmed by the RC
  CommandBuffered    : BOOL;
  /// Frame data
  FrameData           : FrameData;
END_VAR

                  
                

METHOD PROTECTED OnCall
VAR_IN_OUT
  /// Robot assignment of function
  AxesGroup         : AxesGroup; 
END_VAR
                        
                      
END_METHOD
END_FUNCTION_BLOCK

/// Calculate Inverse Kinematic
FUNCTION_BLOCK CalculateInverseKinematicFB EXTENDS RobotLibraryBaseFB
// ------------------------------------------------------------------------- 
//  SRCI Robot Library                                                
// ------------------------------------------------------------------------- 
//                                                                           
//  Object:      CalculateInverseKinematicFB                                       
//  Author:      Thorsten Brach                                                
//  Date:        2024-06-01
//
//  Description:                                              
//   
//                                                                           
//  Copyright: 
//    (C) 2024 Thorsten Brach. All rights reserved                                                                         
//                                                                           
//  Disclaimer:                                                                           
//    This project is provided without any guarantee and can be used for   
//    private and commercial purposes. Any commercial use is at the user’s 
//    own risk and responsibility.
//
// -------------------------------------------------------------------------
VAR_INPUT
  /// Start of the command at the rising edge
  Execute            : BOOL;
  /// cartesian position
  CartesianPosition  : RobotCartesianPosition;
  /// Index of target tool
  /// • 0: Flange (default)
  /// • 1..254: Tool frames
  ToolNo             : USINT;
  /// Index of target frame
  /// • 0: WCS (default)
  /// • 1..254: User frames
  FrameNo            : USINT;  
END_VAR
VAR_OUTPUT
  /// The command has been completed successfully
  Done               : BOOL;
  /// FB is being processed
  Busy               : BOOL;
  /// Command is transferred and confirmed by the RC
  CommandBuffered    : BOOL;
  /// Calculated robot joint position
  JointPosition      : RobotJointPosition;
END_VAR

                  
                

METHOD PROTECTED OnCall
VAR_IN_OUT
  /// Robot assignment of function
  AxesGroup         : AxesGroup; 
END_VAR
                        
                      
END_METHOD
END_FUNCTION_BLOCK

/// Calculate tool (TCP) with four-point method
FUNCTION_BLOCK CalculateToolFB EXTENDS RobotLibraryBaseFB
// ------------------------------------------------------------------------- 
//  SRCI Robot Library                                                
// ------------------------------------------------------------------------- 
//                                                                           
//  Object:      CalculateToolFB                                       
//  Author:      Thorsten Brach                                                
//  Date:        2024-06-01
//
//  Description:                                              
//   
//                                                                           
//  Copyright: 
//    (C) 2024 Thorsten Brach. All rights reserved                                                                         
//                                                                           
//  Disclaimer:                                                                           
//    This project is provided without any guarantee and can be used for   
//    private and commercial purposes. Any commercial use is at the user’s 
//    own risk and responsibility.
//
// -------------------------------------------------------------------------
VAR_INPUT
  /// Start of the command at the rising edge
  Execute            : BOOL;
  /// Define which method should be used to calculate the tool frame
  Mode               : ToolCalculationMode;
  /// Index of target tool
  /// • 0: Flange (default)
  /// • 1..254: Tool frames
  ToolNo             : USINT;
  /// Index of target frame
  /// • 0: WCS (default)
  /// • 1..254: User frames
  FrameNo            : USINT;  
  /// • True: Tool fixed
  /// • False: Tool on flange (default)
  ExternalTCP        : BOOL;
  /// Positions in cartesian coordinates for the tool frame calculation.
  PositionsArray     : ARRAY[0..5] OF RobotCartesianPosition;
END_VAR
VAR_OUTPUT
  /// The command has been completed successfully
  Done               : BOOL;
  /// FB is being processed
  Busy               : BOOL;
  /// Command is transferred and confirmed by the RC
  CommandBuffered    : BOOL;
  /// Tool data
  ToolData           : ToolData;
  /// Maximum error of deviation of the TCP position
  /// from the fix point in world coordinate system
  /// If not supported: • -1
  TCPMaxError       : REAL;
  /// Average error of TCP position from the fix point  in world coordinate system
  /// If not supported: • -1 
  TCPMeanError      : REAL;
END_VAR

                  
                

METHOD PROTECTED OnCall
VAR_IN_OUT
  /// Robot assignment of function
  AxesGroup         : AxesGroup; 
END_VAR
                        
                      
END_METHOD
END_FUNCTION_BLOCK

/// Activate conveyor tracking mode
FUNCTION_BLOCK ActivateConveyorTrackingFB EXTENDS RobotLibraryBaseFB
// ------------------------------------------------------------------------- 
//  SRCI Robot Library                                                
// ------------------------------------------------------------------------- 
//                                                                           
//  Object:      ActivateConveyorTrackingFB                                       
//  Author:      Thorsten Brach                                                
//  Date:        2024-06-01
//
//  Description:                                              
//   
//                                                                           
//  Copyright: 
//    (C) 2024 Thorsten Brach. All rights reserved                                                                         
//                                                                           
//  Disclaimer:                                                                           
//    This project is provided without any guarantee and can be used for   
//    private and commercial purposes. Any commercial use is at the user’s 
//    own risk and responsibility.
//
// -------------------------------------------------------------------------
VAR_INPUT
  /// Set TRUE to change RA power state to "Enabled"
  Enable             : BOOL;
  /// Index of assigned conveyor
  ConveyorNo         : USINT;
  /// Specifies encoder connection setup (at least one option must be supported)
  ConnectionMode     : ConnectionMode;
  /// Relates to "ConnectionMode" 1 – "PLC connected": Value of the encoder connected to the conveyor belt
  PLCEncoderValue    : REAL;
END_VAR

VAR_OUTPUT
  /// TRUE, while the following outputs return valid values:
  /// • TrackingStatusByte
  /// • RCEncoderValue
  Valid              : BOOL;
  /// FB is being processed
  Busy               : BOOL;
  /// Command is transferred and confirmed by the RC
  CommandBuffered    : BOOL;
  /// Receiving of input parameter values has been acknowledged by RC
  ParameterAccepted  : BOOL;
  /// Current status of "ConveyorTracking" according to Table 6-432
  TrackingStatus     : TrackingStatus;
  /// Relates to "ConnectionMode" 1 – "RC connected": Traveled distance of assigned conveyor since ConveyorTracking has been activated (offset)
  RCEncoderValue     : REAL;
END_VAR

                  
                

METHOD Protected OnCall
VAR_IN_OUT
  /// Robot assignment of function
  AxesGroup         : AxesGroup; 
END_VAR
                        
                      
END_METHOD
END_FUNCTION_BLOCK

/// Configure conveyor parameters
FUNCTION_BLOCK ConfigureConveyorFB EXTENDS RobotLibraryBaseFB
// ------------------------------------------------------------------------- 
//  SRCI Robot Library                                                
// ------------------------------------------------------------------------- 
//                                                                           
//  Object:      ConfigureConveyorFB                                       
//  Author:      Thorsten Brach                                                
//  Date:        2024-06-01
//
//  Description:                                              
//   
//                                                                           
//  Copyright: 
//    (C) 2024 Thorsten Brach. All rights reserved                                                                         
//                                                                           
//  Disclaimer:                                                                           
//    This project is provided without any guarantee and can be used for   
//    private and commercial purposes. Any commercial use is at the user’s 
//    own risk and responsibility.
//
// -------------------------------------------------------------------------
VAR_INPUT
  /// Start of the command at the rising edge
  Execute            : BOOL;
  /// Index of assigned conveyor
  ConveyorNo         : USINT;  
  ///Define the origin coordinate system of the conveyor belt, with the X-Axis pointing in the direction of the movement of the conveyor belt.
  ConveyorOrigin     : FrameData;
  /// Define the type of the conveyor
  ConveyorType       : ConveyorType;
  /// Relates to "ConveyorType" "Circular Tracking": Define the radius of the circular conveyor
  Radius             : REAL;
  /// Distance [mm] from the origin of the conveyor belt to the beginning of the "SyncInZone"
  StartDistance      : REAL;
  /// Distance [mm] from the origin of the conveyor belt to the end of the "SyncOutZone"
  EndDistance        : REAL;
  /// Define the length of the "SyncInZone"
  SyncInLength       : REAL;
  /// Define the length of the "SyncOutZone"
  SyncOutLength      : REAL;
END_VAR

VAR_OUTPUT
  /// The command has been completed successfully
  Done               : BOOL;
  /// FB is being processed
  Busy               : BOOL;
  /// Command is transferred and confirmed by the RC
  CommandBuffered    : BOOL;
END_VAR

                  
                

METHOD PROTECTED OnCall
VAR_IN_OUT
  /// Robot assignment of function
  AxesGroup         : AxesGroup; 
END_VAR
                        
                      
END_METHOD
END_FUNCTION_BLOCK

/// Redefine tracking position for conveyor tracking
FUNCTION_BLOCK RedefineTrackingPosFB EXTENDS RobotLibraryBaseFB
// ------------------------------------------------------------------------- 
//  SRCI Robot Library                                                
// ------------------------------------------------------------------------- 
//                                                                           
//  Object:      RedefineTrackingPosFB                                       
//  Author:      Thorsten Brach                                                
//  Date:        2024-06-01
//
//  Description:                                              
//   
//                                                                           
//  Copyright: 
//    (C) 2024 Thorsten Brach. All rights reserved                                                                         
//                                                                           
//  Disclaimer:                                                                           
//    This project is provided without any guarantee and can be used for   
//    private and commercial purposes. Any commercial use is at the user’s 
//    own risk and responsibility.
//
// -------------------------------------------------------------------------
VAR_INPUT
  /// Start of the command at the rising edge
  Execute                : BOOL;
  /// Relates to ListenerID >0:
  ProcessingMode         : ProcessingMode;
  /// Index of assigned conveyor
  ConveyorNo             : USINT;
  /// Relates to ListenerID = 0:
  /// Define initial work piece position relative to the conveyor belt origin:
  /// • Origin (X, Y, Z in mm)
  /// • Orientation (RX, RY, RZ in degree)
  /// For more information refer to chapter 5.5.14.
  InitObjectPosition     : ARRAY[0..5] OF REAL;
  /// Relates to ListenerID = 0:
  /// Travel distance of assigned UCS between work piece detection (InitObjectPosition) and execution of this command.
  TrackingOffset         : REAL;
  /// Relates to ListenerID >0
  /// Start index of real registers containing InitObjectPosition for trigger-based execution.
  StartIndexInitPosition : INT;
  /// Define the index number of the UCS that is assigned to the conveyor by the function "ConveyorTracking".
  /// For more information refer to chapter 5.5.14.
  FrameNo                : USINT;
  /// Relates to ListenerID >0
  /// Index of real register containing TrackingOffset for trigger-based execution
  IndexTrackingOffset    : USINT;
  /// ID of associated trigger function:
  /// • 0: No Trigger (default): No trigger related behavior
  /// • >0: Trigger: o Start executing, when the trigger function with the identical EmitterID is triggered.
  /// Always positive.
  /// For more information, see chapter 5.5.12 Triggers
  ListenerID             :  SINT;
END_VAR

VAR_OUTPUT
  /// The command has been completed successfully
  Done                   : BOOL;
  /// FB is being processed
  Busy                   : BOOL;
  /// Command is transferred and confirmed by the RC
  CommandBuffered        : BOOL;
  /// Receiving of input parameter values has been acknowledged by RC
  ParameterAccepted      : BOOL;
  /// Unique system-generated ID of the "Action" when the function is triggered.
  /// • >0: The "Action" is started by the trigger funcrion with identical FollowID.
  /// • <0: The "Action" is stopped by the trigger function with identical FollowID.
  /// For more information see chapter 5.5.12.4 EmitterID, ListenerID, FollowID and OriginID
  OriginID               : INT;
  /// Relates to ListenerID >0
  /// Number of successful trigger-based command invocations - For more information refer TO chapter 5.5.12.4
  InvocationCounter      : USINT;
END_VAR

                  
                

METHOD PROTECTED OnCall
VAR_IN_OUT
  /// Robot assignment of function
  AxesGroup         : AxesGroup; 
END_VAR
                        
                      
END_METHOD
END_FUNCTION_BLOCK

/// Synchronize robot with conveyor
FUNCTION_BLOCK SyncToConveyorFB EXTENDS RobotLibraryBaseFB
// ------------------------------------------------------------------------- 
//  SRCI Robot Library                                                
// ------------------------------------------------------------------------- 
//                                                                           
//  Object:      SyncToConveyorFB                                       
//  Author:      Thorsten Brach                                                
//  Date:        2024-06-01
//
//  Description:                                              
//   
//                                                                           
//  Copyright: 
//    (C) 2024 Thorsten Brach. All rights reserved                                                                         
//                                                                           
//  Disclaimer:                                                                           
//    This project is provided without any guarantee and can be used for   
//    private and commercial purposes. Any commercial use is at the user’s 
//    own risk and responsibility.
//
// -------------------------------------------------------------------------
VAR_INPUT
  /// Start of the command at the rising edge
  Execute            : BOOL;
  /// Index of assigned conveyor
  ConveyorNo         : USINT;
  /// Define the index number of the UCS that will be assigned to the conveyor.
  /// For more information refer to chapter 5.5.14
  FrameNo            : USINT;
  /// Defines when synchronization starts
  SyncInMode         : SyncInMode;
  /// Relates to "SyncInMode" "After distance" (1) and "After time" (2): Parameter for the synchronization
  /// • "After distance" (1) -  Distance in mm
  /// • "After time" (2) -  Time in ms
  SyncInParameter    : REAL;
  /// Define the maximum adjustment velocity for the robot to catch up to the conveyor belt.
  /// The velocity must be greater than the velocity of the conveyor belt.
  /// • 0 (default): no limit - No conveyor tracking specific limit
  ///                         - RC internal limit applies
  /// • >0: use limit         - Conveyor tracking specific limit applies
  MaxVelocity        : REAL;
  /// Define the maximum adjustment acceleration for the robot to catch up to the conveyor belt.
  /// • 0 (default): no limit - No conveyor tracking specific limit
  ///                         - RC internal limit applies
  /// • >0: use limit         - Conveyor tracking specific limit applies
  MaxAcceleration    : REAL;
  /// ID of associated trigger function:
  /// • 0: No Trigger (default): No trigger related behavior
  /// • >0: Trigger:  Start executing, when the trigger function with the identical EmitterID is triggered.
  /// Always positive.
  /// For more information, see chapter 5.5.12 Triggers
  ListenerID         : SINT;
END_VAR

VAR_OUTPUT
  /// FB is being processed
  Busy               : BOOL;
  /// Command is transferred and confirmed by the RC
  CommandBuffered    : BOOL;
  /// TRUE, while SyncToConveyor is enabled and processing input parameters
  Enabled            : BOOL;
  /// The command takes control of the motion of the according axis group
  Active             : BOOL;
  /// The command was aborted by another command.
  CommandAborted     : BOOL;
  /// Receiving of input parameter values has been acknowledged by RC
  ParameterAccepted  : BOOL;
  /// The TCP is in synchronization with the object on the conveyor belt.
  InSync             : BOOL;
  /// Unique system-generated ID of the "Action" when the function is triggered.
  /// • >0: The "Action" is started by the trigger function with identical FollowID.
  /// • <0: The "Action" is stopped by the trigger function with identical FollowID.
  /// For more information see chapter 5.5.12.4 EmitterID, ListenerID, FollowID and OriginID
  OriginID           : INT;
  /// Relates to ListenerID >0
  /// Number of successful trigger -based command invocations
  /// For more information refer to chapter 5.5.12.4.
  InvocationCounter  : USINT;
END_VAR

                  
                

METHOD PROTECTED OnCall
VAR_IN_OUT
  /// Robot assignment of function
  AxesGroup         : AxesGroup; 
END_VAR
                        
                      
END_METHOD
END_FUNCTION_BLOCK

/// Enables the RC to apply user defined force/ torque through RA’s TCP movement
FUNCTION_BLOCK ForceControlFB EXTENDS RobotLibraryBaseFB
// ------------------------------------------------------------------------- 
//  SRCI Robot Library                                                
// ------------------------------------------------------------------------- 
//                                                                           
//  Object:      ForceControlFB                                       
//  Author:      Thorsten Brach                                                
//  Date:        2024-06-01
//
//  Description:                                              
//   
//                                                                           
//  Copyright: 
//    (C) 2024 Thorsten Brach. All rights reserved                                                                         
//                                                                           
//  Disclaimer:                                                                           
//    This project is provided without any guarantee and can be used for   
//    private and commercial purposes. Any commercial use is at the user’s 
//    own risk and responsibility.
//
// -------------------------------------------------------------------------
VAR_INPUT
  /// Start of the command at the rising edge
  Execute            : BOOL;
  /// Defines type of reference of Force and Torque (at least one option must be supported)
  ReferenceType      : ReferenceType;
  /// Relates to ConnectionMode 1 and 2 (Sensor connected to PLC).
  /// Currently applied force and torque detected by sensor according to ReferenceType, ToolNo and FrameNo.
  /// • [0]: X-Axis
  /// • [1]: Y-Axis
  /// • [2]: Z- Axis
  /// • [3]: Rotation around X-Axis (RX)
  /// • [4]: Rotation around Y-Axis (RY)
  /// • [5]: Rotation around Z- Axis (RZ)
  SensorValue        : ARRAY[0..5] OF REAL;
  /// Relates to ReferenceType 0 (Tool) and 1 (Frame):
  /// Force and torque to be applied by robot arm according to ReferenceType, ToolNo and FrameNo:
  /// • [0]: X-Axis
  /// • [1]: Y-Axis
  /// • [2]: Z- Axis
  /// • [3]: Rotation around X-Axis (RX)
  /// • [4]: Rotation around Y-Axis (RY)
  /// • [5]: Rotation around Z- Axis (RZ)
  /// Set TargetValue <>-99999.9999 (default) to define setpoint
  TargetValue        : ARRAY[0..5] OF REAL;
  /// Index of tool
  /// •      0: Flange (default)
  /// • 1..254: Tool frames
  ToolNo             : USINT;
  /// Define the index number of the UCS that will be assigned to the conveyor.
  /// For more information refer to chapter 5.5.14
  FrameNo            : USINT;
  /// Specifies encoder connection setup according to Table 6-713 (at least one option must be supported) 
  ConnectionMode     : SensorConnectionMode;
  /// Position of sensor relative to flange (FixedSensor FALSE) or relative to WCS (FixedSensor TRUE)
  /// • [0]: X-Axis
  /// • [1]: Y-Axis
  /// • [2]: Z- Axis
  /// • [3]: Rotation around X-Axis (RX)
  /// • [4]: Rotation around Y-Axis (RY)
  /// • [5]: Rotation around Z- Axis (RZ)
  SensorFrame        : ARRAY[0..5] OF REAL;
  /// Index of payload data containing mass, center of gravity, orientation and inertia relative to SensorFrame.
  /// Required to calibrate system for setting up gravity compensation and sensor offset.
  CalibrationData    : USINT;
  /// Tolerance of TargetValue within which currently applied force/torque will return ForceStatus "Specified force/torque reached" TRUE.
  TargetWindow       : REAL;
  /// Define axes whose position may be adjusted by the robot to apply specified force according to Table 6-711.
  CompliantAxes      : BYTE;
  /// Maximum allowed TCP velocity for compliant axes in % of nominal velocity.
  /// •   0% (default): no limit - RC internal limit applies
  /// •  >0% use limit -  Specified limit applies
  /// • 100% use maximal reference velocity
  /// For more information on nominal dynamics see chapter 5.5.7 Robot dynamics 
  MaxVelocity        : REAL;
  /// Maximum allowed cartesian deviation according to ReferenceType, ToolNo and FrameNo.
  /// Set 0 (default) to not specify a limit in this axis direction.
  /// • [0]: Deviation in X-Direction in mm
  /// • [1]: Deviation in Y- direction in mm
  /// • [2]: Deviation in Z- direction in mm
  /// • [3]: Deviation in RX- direction in °
  /// • [4]: Deviation in RY- direction in °
  /// • [5]: Deviation in RZ- direction in °
  MaxDeviation       : ARRAY [0..5] OF REAL;
  /// Defines reaction in case ForceControl reports error during its execution
  /// Processing of active move command is continued without active ForceControl
  ErrorReaction      : ErrorReaction;
  /// Relates to ErrorReaction 0 (Abort and move). Defines type of reference coordinate system of ErrorVector
  ErrorReferenceType : ReferenceType;
  /// Relates to ErrorReaction 0 (Abort and move). Vector defining robot’s movement in case of
  /// incoming error according to ErrorReferenceType, ErrorToolNo and ErrorFrameNo.
  /// • [0]: X-Axis
  /// • [1]: Y-Axis
  /// • [2]: Z- Axis
  /// • [3]: Rotation around X-Axis (RX)
  /// • [4]: Rotation around Y-Axis (RY)
  /// • [5]: Rotation around Z-Axis (RZ)
  ErrorVector        : ARRAY [0..5] OF REAL;
  /// Relates to ErrorReaction 0 (Abort and move). Index of tool.
  /// • 0 (default): Flange
  /// • 1..254: Tool frames
  ErrorToolNo        : USINT;
  /// Relates to ErrorReferenceType 1 (Frame)
  /// •      0: WCS (default)
  /// • 1..254: User frames
  ErrorFrameNo       : USINT;
  /// Defines sensor positioning:
  /// • FALSE (default): Sensor mounted on flange
  /// • TRUE: Sensor fixed
  FixedSensor        : BOOL;
END_VAR

VAR_OUTPUT
  /// TRUE, while the following outputs return valid values:
  /// - ForceStatus
  Valid              : BOOL;
  /// FB is being processed
  Busy               : BOOL;
  /// Command is transferred and confirmed by the RC
  CommandBuffered    : BOOL;
  /// Receiving of input parameter values has been acknowledged by RC
  ParameterAccepted  : BOOL;
  /// Current status of ForceControl and ForceLimit (chapter 6.5.25) according to Table 6-712
  ForceStatus        : ForceStatus;
END_VAR

                  
                

METHOD PROTECTED OnCall
VAR_IN_OUT
  /// Robot assignment of function
  AxesGroup         : AxesGroup; 
END_VAR
                        
                      
END_METHOD
END_FUNCTION_BLOCK

/// Commands specified reaction from RA when defined force/torque detected
FUNCTION_BLOCK ForceLimitFB EXTENDS RobotLibraryBaseFB
// ------------------------------------------------------------------------- 
//  SRCI Robot Library                                                
// ------------------------------------------------------------------------- 
//                                                                           
//  Object:      ForceLimitFB                                       
//  Author:      Thorsten Brach                                                
//  Date:        2024-06-01
//
//  Description:                                              
//   
//                                                                           
//  Copyright: 
//    (C) 2024 Thorsten Brach. All rights reserved                                                                         
//                                                                           
//  Disclaimer:                                                                           
//    This project is provided without any guarantee and can be used for   
//    private and commercial purposes. Any commercial use is at the user’s 
//    own risk and responsibility.
//
// -------------------------------------------------------------------------
VAR_INPUT
  /// Start of the command at the rising edge
  Execute            : BOOL;
  /// Defines type of reference of Force and Torque (at least one option must be supported)
  ReferenceType      : ReferenceType;
  /// Relates to ConnectionMode 1 and 2 (Sensor connected to PLC).
  /// Currently applied force and torque detected by sensor according to ReferenceType, ToolNo and FrameNo.
  /// • [0]: X-Axis
  /// • [1]: Y-Axis
  /// • [2]: Z- Axis
  /// • [3]: Rotation around X-Axis (RX)
  /// • [4]: Rotation around Y-Axis (RY)
  /// • [5]: Rotation around Z- Axis (RZ)
  SensorValue        : ARRAY[0..5] OF REAL;
  /// Index of tool
  /// •      0: Flange (default)
  /// • 1..254: Tool frames
  ToolNo             : USINT;
  /// Define the index number of the UCS that will be assigned to the conveyor.
  /// For more information refer to chapter 5.5.14
  FrameNo            : USINT;
  /// Maximal allowed force and torque detected by the sensor according to ReferenceType and ToolNo/FrameNo before robot reacts according to ReactionMode.
  /// Set value <>0 (default) to monitor coordinate axes
  /// • [0]: X-Axis
  /// • [1]: Y-Axis
  /// • [2]: Z- Axis
  /// • [3]: Rotation around X-Axis (RX)
  /// • [4]: Rotation around Y-Axis (RY)
  /// • [5]: Rotation around Z- Axis (RZ)
  ForceLimit        : ARRAY[0..5] OF REAL;
  /// Specifies encoder connection setup according to Table 6-713 (at least one option must be supported) 
  ConnectionMode    : SensorConnectionMode;
  /// Position of sensor relative to flange (FixedSensor FALSE) or relative to WCS (FixedSensor TRUE)
  /// • [0]: X-Axis
  /// • [1]: Y-Axis
  /// • [2]: Z- Axis
  /// • [3]: Rotation around X-Axis (RX)
  /// • [4]: Rotation around Y-Axis (RY)
  /// • [5]: Rotation around Z- Axis (RZ)
  SensorFrame        : ARRAY[0..5] OF REAL;
  /// Index of payload data containing mass, center of gravity, orientation and inertia relative to SensorFrame.
  /// Required to calibrate system for setting up gravity compensation and sensor offset.
  CalibrationData    : USINT;
  /// Defines sensor positioning:
  /// • FALSE (default): Sensor mounted on flange
  /// • TRUE: Sensor fixed
  FixedSensor        : BOOL;
  /// ID of Action that will be executed when this command is active
  /// • >0: Start Action        - Start executing the Action function with the identical ListenerID.
  /// • <0: Stop Action         - Stop executing the Action function with the identical ListenerID.
  /// •  0: Undefined (default) - If no EmitterID is defined, the function returns an error message
  /// For more information see chapter 5.5.12.4
  EmitterID          : SINT;  
END_VAR

VAR_OUTPUT
  /// TRUE, while the following outputs return valid values
  Valid              : BOOL;
  /// FB is being processed
  Busy               : BOOL;
  /// Command is transferred and confirmed by the RC
  CommandBuffered    : BOOL;
  /// Receiving of input parameter values has been acknowledged by RC
  ParameterAccepted  : BOOL;
  /// Current status of ForceControl and ForceLimit (chapter 6.5.25) according to Table 6-712
  ForceStatus        : ForceStatus;
  /// Relates to EmitterID <> 0: Unique system-generated ID of the trigger function when the function is called by user.
  /// For more information see chapter 5.5.12.4.
  FollowID           : DINT;
END_VAR

                  
                

METHOD PROTECTED OnCall
VAR_IN_OUT
  /// Robot assignment of function
  AxesGroup         : AxesGroup; 
END_VAR
                        
                      
END_METHOD
END_FUNCTION_BLOCK

/// Read actual force/torque at TCP
FUNCTION_BLOCK ReadActualForceFB EXTENDS RobotLibraryBaseFB
// ------------------------------------------------------------------------- 
//  SRCI Robot Library                                                
// ------------------------------------------------------------------------- 
//                                                                           
//  Object:      ReadActualForceFB                                       
//  Author:      Thorsten Brach                                                
//  Date:        2024-06-01
//
//  Description:                                              
//   
//                                                                           
//  Copyright: 
//    (C) 2024 Thorsten Brach. All rights reserved                                                                         
//                                                                           
//  Disclaimer:                                                                           
//    This project is provided without any guarantee and can be used for   
//    private and commercial purposes. Any commercial use is at the user’s 
//    own risk and responsibility.
//
// -------------------------------------------------------------------------
VAR_INPUT
  /// Start of the command at the rising edge
  Execute            : BOOL;
  /// Processing Mode
  ProcessingMode      : ProcessingMode;
  /// Defines type of reference of Force and Torque (at least one option must be supported )
  ReferenceType       : ReferenceType;
  /// Index of tool
  /// •      0: Flange (default)
  /// • 1..254: Tool frames
  ToolNo             : USINT;
  /// Define the index number of the UCS that will be assigned to the conveyor.
  /// For more information refer to chapter 5.5.14
  FrameNo            : USINT;
  /// Index of payload data containing mass, center of gravity, orientation and inertia relative to SensorFrame.
  /// Required to calibrate system for setting up gravity compensation and sensor offset.
  CalibrationData    : USINT;
  /// ID of associated trigger function:
  /// • 0: Immediately (default) - Start executing this function immediately.
  /// • >0: Trigger -  Start executing, when the trigger function with the identical EmitterID is triggered.
  /// Always positive.
  /// For more information, see chapter 5.5.12 Triggers
  ListenerID         : SINT;
 
END_VAR

VAR_OUTPUT
  /// TRUE, when command has been completed successfully.
  Done               : BOOL;
  /// TRUE, while the following outputs return valid values:
  /// - ActualForce
  Valid              : BOOL;
  /// FB is being processed
  Busy               : BOOL;
  /// Command is transferred and confirmed by the RC
  CommandBuffered    : BOOL;
  /// Receiving of input parameter values has been acknowledged by RC
  ParameterAccepted  : BOOL;
  /// Currently detected force and torque according to ReferenceType, ToolNo and FrameNo.
  /// • [0]: X-Axis
  /// • [1]: Y-Axis
  /// • [2]: Z- Axis
  /// • [3]: Rotation around X-Axis (RX)
  /// • [4]: Rotation around Y-Axis (RY)
  /// • [5]: Rotation around Z- Axis (RZ)
  ActualForce        : ARRAY[0..5] OF REAL;
  /// Unique system-generated ID of the "Action" when the function is triggered.
  /// • >0: The "Action" is started by the trigger function with identical FollowID.
  /// • <0: The "Action" is stopped by the trigger function with identical FollowID.
  /// For more information see chapter 5.5.12.4 EmitterID, ListenerID, FollowID and OriginID
  OriginID           : INT;
  /// Relates to ListenerID >0
  /// Number of successful trigger -based command invocations
  /// For more information refer to chapter 5.5.12.4.
  InvocationCounter  : USINT;
  
END_VAR

                  
                

METHOD PROTECTED OnCall
VAR_IN_OUT
  /// Robot assignment of function
  AxesGroup         : AxesGroup; 
END_VAR
                        
                      
END_METHOD
END_FUNCTION_BLOCK

/// Continue interrupted path
FUNCTION_BLOCK GroupContinueFB EXTENDS RobotLibraryBaseFB
// ------------------------------------------------------------------------- 
//  SRCI Robot Library                                                
// ------------------------------------------------------------------------- 
//                                                                           
//  Object:      GroupContinueFB                                       
//  Author:      Thorsten Brach                                                
//  Date:        2024-06-01
//
//  Description:                                              
//   
//                                                                           
//  Copyright: 
//    (C) 2024 Thorsten Brach. All rights reserved                                                                         
//                                                                           
//  Disclaimer:                                                                           
//    This project is provided without any guarantee and can be used for   
//    private and commercial purposes. Any commercial use is at the user’s 
//    own risk and responsibility.
//
// -------------------------------------------------------------------------
VAR_INPUT
  /// Start of the command at the rising edge
  Execute            : BOOL;
END_VAR
VAR_OUTPUT
  /// The command has been completed successfully
  Done               : BOOL;
  /// FB is being processed
  Busy               : BOOL;
  /// Command is transferred and confirmed by the RC
  CommandBuffered    : BOOL;
END_VAR

                  
                

METHOD PROTECTED OnCall
VAR_IN_OUT
  /// Robot assignment of function
  AxesGroup         : AxesGroup; 
END_VAR
                        
                      
END_METHOD
END_FUNCTION_BLOCK

/// Interrupt active movement, possible to continue movement
FUNCTION_BLOCK GroupInterruptFB EXTENDS RobotLibraryBaseFB
// ------------------------------------------------------------------------- 
//  SRCI Robot Library                                                
// ------------------------------------------------------------------------- 
//                                                                           
//  Object:      GroupInterruptFB                                       
//  Author:      Thorsten Brach                                                
//  Date:        2024-06-01
//
//  Description:                                              
//   
//                                                                           
//  Copyright: 
//    (C) 2024 Thorsten Brach. All rights reserved                                                                         
//                                                                           
//  Disclaimer:                                                                           
//    This project is provided without any guarantee and can be used for   
//    private and commercial purposes. Any commercial use is at the user’s 
//    own risk and responsibility.
//
// -------------------------------------------------------------------------
VAR_INPUT
  /// Start of the command at the rising edge
  Execute            : BOOL;
END_VAR

VAR_OUTPUT
  /// The command has been completed successfully
  Done               : BOOL;
  /// FB is being processed
  Busy               : BOOL;
  /// Command is transferred and confirmed by the RC
  CommandBuffered    : BOOL;
  /// The command takes control of the motion of the according axis group.
  Active             : BOOL;
END_VAR

                  
                

METHOD PROTECTED OnCall
VAR_IN_OUT
  /// Robot assignment of function
  AxesGroup         : AxesGroup; 
END_VAR
                        
                      
END_METHOD
END_FUNCTION_BLOCK

/// Jog robot manually
FUNCTION_BLOCK GroupJogFB EXTENDS RobotLibraryBaseFB
// ------------------------------------------------------------------------- 
//  SRCI Robot Library                                                
// ------------------------------------------------------------------------- 
//                                                                           
//  Object:      GroupJogFB                                       
//  Author:      Thorsten Brach                                                
//  Date:        2024-06-01
//
//  Description:                                              
//   
//                                                                           
//  Copyright: 
//    (C) 2024 Thorsten Brach. All rights reserved                                                                         
//                                                                           
//  Disclaimer:                                                                           
//    This project is provided without any guarantee and can be used for   
//    private and commercial purposes. Any commercial use is at the user’s 
//    own risk and responsibility.
//
// -------------------------------------------------------------------------
VAR_INPUT
  /// Activate jog command
  Enable                 : BOOL;
  /// Specifies in which mode the robot is jogged
  Mode                   : JogMode;
  /// Velocity in % of monitoring speed or ReferenceVelocity, depending on the currently active operation mode 
  /// (T1 External/T2 External: Monitoring speed; Automatic External: ReferenceVelocity )
  /// •    0%: No movement of the robot
  /// •   10%: default
  /// • ≤100%: use input parameter value
  Override               : REAL;
  /// Change to jog and define direction according to Mode. See Table 6-223
  Control                : JogControl;
  /// Relates to Mode 0 (JogFrame) and 1 (JogTool) Index of tool
  /// •      0: Flange (default):
  /// • 1..254: Tool frames
  ToolNo                 : USINT;
  /// Relates to Mode 0 (JogFrame) Index of frame
  /// •      0: WCS (default)
  /// • 1..254: User frames
  FrameNo                : USINT;
  /// Increments for jogging translational axes for defined distance
  /// •  0: Incremental mode OFF (default) - Movement is active until "Control" is reset, or error occurs.
  /// • >0: Incremental mode ON            - Movement is active until distance defined by input value is reached without changes to "Control", "Control" is reset, or error occurs
  IncrementalTranslation : REAL;
  /// Increments for jogging rotational axes for defined distance
  /// • 0: Incremental mode OFF (default) - Movement is active until "Control" is reset, or error occurs.
  /// • >0 Incremental mode ON:           - Movement is active until distance defined by input value is reached without changes to "Control", "Control" is reset, or error occurs
  IncrementalRotation    : REAL;
END_VAR

VAR_OUTPUT
  /// Relates to Incremental mode ON: TRUE, when robot’s TCP or axes have traversed distance of "IncrementalTranslation" or "IncrementalRotation"
  DistanceReached        : BOOL;
  /// FB is being processed
  Busy                   : BOOL;
  /// Command is transferred and confirmed by the RC
  CommandBuffered        : BOOL;
  /// TRUE while GroupJog is enabled
  Enabled                : BOOL;
  /// The command takes control of the motion of the according axis group
  Active                 : BOOL;
  /// The active movement was aborted by another command
  CommandAborted         : BOOL;
  /// Receiving of input parameter values has been acknowledged by RC
  ParameterAccepted      : BOOL;
END_VAR

                  
                

METHOD PROTECTED OnCall
VAR_IN_OUT
  /// Robot assignment of function
  AxesGroup         : AxesGroup; 
END_VAR
                        
                      
END_METHOD
END_FUNCTION_BLOCK

/// Acknowledgement all pending errors
FUNCTION_BLOCK GroupResetFB EXTENDS RobotLibraryBaseFB
// ------------------------------------------------------------------------- 
//  SRCI Robot Library                                                
// ------------------------------------------------------------------------- 
//                                                                           
//  Object:      GroupResetFB                                       
//  Author:      Thorsten Brach                                                
//  Date:        2024-06-01
//
//  Description:                                              
//   
//                                                                           
//  Copyright: 
//    (C) 2024 Thorsten Brach. All rights reserved                                                                         
//                                                                           
//  Disclaimer:                                                                           
//    This project is provided without any guarantee and can be used for   
//    private and commercial purposes. Any commercial use is at the user’s 
//    own risk and responsibility.
//
// -------------------------------------------------------------------------
VAR_INPUT
  /// Start of the command at the rising edge
  Execute         : BOOL;
END_VAR

VAR_OUTPUT
  /// The command has been completed successfully
  Done            : BOOL;
  /// FB is being processed
  Busy            : BOOL;
  /// Command is transferred and confirmed by the RC
  CommandBuffered : BOOL;
END_VAR

                  
                

METHOD PROTECTED OnCall
VAR_IN_OUT
  /// Robot assignment of function
  AxesGroup         : AxesGroup; 
END_VAR
                        
                      
END_METHOD
END_FUNCTION_BLOCK

/// Abort actual movement and delete buffer
FUNCTION_BLOCK GroupStopFB EXTENDS RobotLibraryBaseFB
// ------------------------------------------------------------------------- 
//  SRCI Robot Library                                                
// ------------------------------------------------------------------------- 
//                                                                           
//  Object:      GroupStopFB                                       
//  Author:      Thorsten Brach                                                
//  Date:        2024-06-01
//
//  Description:                                              
//   
//                                                                           
//  Copyright: 
//    (C) 2024 Thorsten Brach. All rights reserved                                                                         
//                                                                           
//  Disclaimer:                                                                           
//    This project is provided without any guarantee and can be used for   
//    private and commercial purposes. Any commercial use is at the user’s 
//    own risk and responsibility.
//
// -------------------------------------------------------------------------
VAR_INPUT
  /// Start of the command at the rising edge
  Execute            : BOOL;
END_VAR

VAR_OUTPUT
  /// The command has been completed successfully
  Done               : BOOL;
  /// FB is being processed
  Busy               : BOOL;
  /// Command is transferred and confirmed by the RC
  CommandBuffered    : BOOL;
  /// Frame index
  AbortedSequence    : SequenceFlag;
END_VAR

                  
                

METHOD PROTECTED OnCall
VAR_IN_OUT
  /// Robot assignment of function
  AxesGroup         : AxesGroup; 
END_VAR
                        
                      
END_METHOD
END_FUNCTION_BLOCK

/// Automatic detection of load data
FUNCTION_BLOCK LoadMeasurementAutomaticFB EXTENDS RobotLibraryBaseFB
// ------------------------------------------------------------------------- 
//  SRCI Robot Library                                                
// ------------------------------------------------------------------------- 
//                                                                           
//  Object:      LoadMeasurementAutomaticFB                                       
//  Author:      Thorsten Brach                                                
//  Date:        2024-06-01
//
//  Description:                                              
//   
//                                                                           
//  Copyright: 
//    (C) 2024 Thorsten Brach. All rights reserved                                                                         
//                                                                           
//  Disclaimer:                                                                           
//    This project is provided without any guarantee and can be used for   
//    private and commercial purposes. Any commercial use is at the user’s 
//    own risk and responsibility.
//
// -------------------------------------------------------------------------
VAR_INPUT
  /// Start of the command at the rising edge
  Execute            : BOOL;
  /// Define which method should be used to measure the load data
  Mode               : LoadMeasurementMode;
  /// Parameter which determines the behavior towards the previously sent and still active or buffered commands.
  AbortingMode       : AbortingMode;
  /// Define which mass is expected as a result of the load measurement
  Mass               : REAL;
  /// Define the area for the allowed motion of the Joint 3. 
  /// The order of the two limit values does not matter. 
  /// Only considered with "Mode" = 0, 2.
  Area_J3            : ARRAY[0..1] OF REAL;
  /// Define the area for the allowed motion of the Joint 4. 
  /// The order of the two limit values does not matter. 
  /// Only considered with "Mode" = 0, 2.
  Area_J4            : ARRAY[0..1] OF REAL;
  /// Define the area for the allowed motion of the Joint 5. 
  /// The order of the two limit values does not matter. 
  /// Only considered with "Mode" = 0, 2.
  Area_J5            : ARRAY[0..1] OF REAL;
  /// Define the area for the allowed motion of the Joint 6. 
  /// The order of the two limit values does not matter. 
  /// Only considered with "Mode" = 0, 2.
  Area_J6            : ARRAY[0..1] OF REAL;
  /// Define the first position for the load measurement.
  /// Only considered with "Mode" = 0, 1.
  Position_1         : RobotJointPosition;
  /// Define the second position for the load measurement.
  /// Only considered with "Mode" = 3.
  Position_2         : RobotJointPosition;
  /// Define the configuration angle for the load measurement.
  /// Only considered with "Mode" = 1.
  ConfigurationAngle : REAL;
  /// Defines the target sequence in which the command will be executed
  SequenceFlag       : SequenceFlag;
END_VAR
VAR_OUTPUT
  ///The command has been completed successfully
  Done               : BOOL;
  /// FB is being processed
  Busy               : BOOL;
  /// Command is transferred and confirmed by the RC
  CommandBuffered    : BOOL;  
  /// The command takes control of the motion of the according axis group.
  Active             : BOOL;
  /// The command was aborted by another command.
  CommandAborted     : BOOL;
  /// TRUE, while command is interrupted during execution and can be continued.
  CommandInterrupted : BOOL;
  /// FB is returning a unique ID for the cal led measurement.
  MeasuringID        : UINT;
  /// Measured load data (see chapter 5.5.6.4)
  LoadData           : LoadData;
END_VAR

                  
                

METHOD PROTECTED OnCall
VAR_IN_OUT
  /// Robot assignment of function
  AxesGroup         : AxesGroup; 
END_VAR
                        
                      
END_METHOD
END_FUNCTION_BLOCK

/// Sequential detection of load data
FUNCTION_BLOCK LoadMeasurementSequentialFB EXTENDS RobotLibraryBaseFB
// ------------------------------------------------------------------------- 
//  SRCI Robot Library                                                
// ------------------------------------------------------------------------- 
//                                                                           
//  Object:      LoadMeasurementSequentialFB                                       
//  Author:      Thorsten Brach                                                
//  Date:        2024-06-01
//
//  Description:                                              
//   
//                                                                           
//  Copyright: 
//    (C) 2024 Thorsten Brach. All rights reserved                                                                         
//                                                                           
//  Disclaimer:                                                                           
//    This project is provided without any guarantee and can be used for   
//    private and commercial purposes. Any commercial use is at the user’s 
//    own risk and responsibility.
//
// -------------------------------------------------------------------------
VAR_INPUT
  /// Start of the command at the rising edge
  Execute            : BOOL;
  /// Processing mode
  ProcessingMode     : ProcessingMode;
  /// Define which step of the load estimation should be executed:
  Mode               : LoadMeasurementSteps;
  /// Define which mass is expected as a result of the load measurement
  Mass               : REAL;
  /// Defines the target sequence in which the command will be executed
  SequenceFlag       : SequenceFlag;
END_VAR

VAR_OUTPUT
  ///The command has been completed successfully
  Done               : BOOL;
  /// FB is being processed
  Busy               : BOOL;
  /// Command is transferred and confirmed by the RC
  CommandBuffered    : BOOL;  
  /// The command takes control of the motion of the according axis group.
  Active             : BOOL;
  /// The command was aborted by another command.
  CommandAborted     : BOOL;
  /// TRUE, while command is interrupted during execution and can be continued.
  CommandInterrupted : BOOL;
  /// FB is returning a unique ID for the cal led measurement.
  MeasuringID        : UINT;
  /// Measured load data (see chapter 5.5.6.4)
  LoadData           : LoadData;
END_VAR

                  
                

METHOD PROTECTED OnCall
VAR_IN_OUT
  /// Robot assignment of function
  AxesGroup         : AxesGroup; 
END_VAR
                        
                      
END_METHOD
END_FUNCTION_BLOCK

/// Abort triggering of Position, measuring input
FUNCTION_BLOCK AbortMeasuringInputFB EXTENDS RobotLibraryBaseFB
// ------------------------------------------------------------------------- 
//  SRCI Robot Library                                                
// ------------------------------------------------------------------------- 
//                                                                           
//  Object:      AbortMeasuringInputFB                                       
//  Author:      Thorsten Brach                                                
//  Date:        2024-06-01
//
//  Description:                                              
//   
//                                                                           
//  Copyright: 
//    (C) 2024 Thorsten Brach. All rights reserved                                                                         
//                                                                           
//  Disclaimer:                                                                           
//    This project is provided without any guarantee and can be used for   
//    private and commercial purposes. Any commercial use is at the user’s 
//    own risk and responsibility.
//
// -------------------------------------------------------------------------
VAR_INPUT
  /// Start of the command at the rising edge
  Execute            : BOOL;
  /// Define an active measurement that is to be aborted.
  /// •  0: Abort all existing measurement
  /// • >0: Abort the measurement with the specific MeasuringID
  MeasuringID        : UINT;
END_VAR
VAR_OUTPUT
  ///The command has been completed successfully
  Done               : BOOL;
  /// FB is being processed
  Busy               : BOOL;
  /// Command is transferred and confirmed by the RC
  CommandBuffered    : BOOL;  
END_VAR

                  
                

METHOD PROTECTED OnCall
VAR_IN_OUT
  /// Robot assignment of function
  AxesGroup         : AxesGroup; 
END_VAR
                        
                      
END_METHOD
END_FUNCTION_BLOCK

/// Capture trigger Position, measuring input
FUNCTION_BLOCK MeasuringInputFB EXTENDS RobotLibraryBaseFB
// ------------------------------------------------------------------------- 
//  SRCI Robot Library                                                
// ------------------------------------------------------------------------- 
//                                                                           
//  Object:      MeasuringInputFB                                       
//  Author:      Thorsten Brach                                                
//  Date:        2024-06-01
//
//  Description:                                              
//   
//                                                                           
//  Copyright: 
//    (C) 2024 Thorsten Brach. All rights reserved                                                                         
//                                                                           
//  Disclaimer:                                                                           
//    This project is provided without any guarantee and can be used for   
//    private and commercial purposes. Any commercial use is at the user’s 
//    own risk and responsibility.
//
// -------------------------------------------------------------------------
VAR_INPUT
  /// Start of the command at the rising edge
  Execute            : BOOL;
  /// Type of measurement (at least one option must be supported):
  MeasuringMode      : MeasuringIoMode;
  /// Specifies the desired digital input register. 
  /// More information about the different periphery register can be found in chapter 6.4
  Index              : USINT;
  ///Specifies the desired bit in the digital input register, that should be read. 
  /// More information about the different periphery register can be found in chapter 6.4.
  BitNumber          : USINT;
END_VAR

VAR_OUTPUT
  ///The command has been completed successfully
  Done               : BOOL;
  /// FB is being processed
  Busy               : BOOL;
  /// Command is transferred and confirmed by the RC
  CommandBuffered    : BOOL;  
  /// FB is returning a unique ID for the cal led measurement.
  MeasuringID        : UINT;
  /// Measured robot position value at the rising edge of the digital input in selected coordinate systems (see input parameters ToolNo and FrameNo).
  Measurings         : ARRAY[1..2] OF MeasuringInputResult;
END_VAR

                  
                

METHOD PROTECTED OnCall
VAR_IN_OUT
  /// Robot assignment of function
  AxesGroup         : AxesGroup; 
END_VAR
                        
                      
END_METHOD
END_FUNCTION_BLOCK

/// Activate/Deactivate functionality to avoid singularities
FUNCTION_BLOCK AvoidSingularityFB EXTENDS RobotLibraryBaseFB
// ------------------------------------------------------------------------- 
//  SRCI Robot Library                                                
// ------------------------------------------------------------------------- 
//                                                                           
//  Object:      AvoidSingularityFB                                       
//  Author:      Thorsten Brach                                                
//  Date:        2024-06-01
//
//  Description:                                              
//   
//                                                                           
//  Copyright: 
//    (C) 2024 Thorsten Brach. All rights reserved                                                                         
//                                                                           
//  Disclaimer:                                                                           
//    This project is provided without any guarantee and can be used for   
//    private and commercial purposes. Any commercial use is at the user’s 
//    own risk and responsibility.
//
// -------------------------------------------------------------------------
VAR_INPUT
  /// Set TRUE to activate avoid singularity mode
  Enable            : BOOL;
  /// Define in which way the singularity should be avoided
  Mode              : SingularityAvoidanceMode;
END_VAR

VAR_OUTPUT
  /// FB is being processed
  Busy              : BOOL;
  /// Command is transferred and confirmed by the RC
  CommandBuffered   : BOOL;
  /// TRUE while AvoidSingularity is active
  Enabled           : BOOL;
  /// Receiving of input parameter values has been acknowledged by RC
  ParameterAccepted : BOOL;
END_VAR

                  
                

METHOD PROTECTED OnCall
VAR_IN_OUT
  /// Robot assignment of function
  AxesGroup         : AxesGroup; 
END_VAR
                        
                      
END_METHOD
END_FUNCTION_BLOCK

/// Change actual speed override
FUNCTION_BLOCK ChangeSpeedOverrideFB EXTENDS RobotLibraryBaseFB
// ------------------------------------------------------------------------- 
//  SRCI Robot Library                                                
// ------------------------------------------------------------------------- 
//                                                                           
//  Object:      ChangeSpeedOverrideFB                                       
//  Author:      Thorsten Brach                                                
//  Date:        2024-06-01
//
//  Description:                                              
//   
//                                                                           
//  Copyright: 
//    (C) 2024 Thorsten Brach. All rights reserved                                                                         
//                                                                           
//  Disclaimer:                                                                           
//    This project is provided without any guarantee and can be used for   
//    private and commercial purposes. Any commercial use is at the user’s 
//    own risk and responsibility.
//
// -------------------------------------------------------------------------
VAR_INPUT
  /// Start of the command at the rising edge
  Execute         : BOOL;
  /// Set value for override
  /// • 0% No movement of the robot
  /// • 10% default
  /// • ≤100%: use input parameter value
  Override        : REAL;
END_VAR

VAR_OUTPUT
  /// The command has been completed successfully
  Done            : BOOL;
  /// FB is being processed
  Busy            : BOOL;
  /// Command is transferred and confirmed by the RC
  CommandBuffered : BOOL;
END_VAR

                  
                

METHOD PROTECTED OnCall
VAR_IN_OUT
  /// Robot assignment of function
  AxesGroup         : AxesGroup; 
END_VAR
                        
                      
END_METHOD
END_FUNCTION_BLOCK

/// Turn on/off the collision detection
FUNCTION_BLOCK CollisionDetectionFB EXTENDS RobotLibraryBaseFB
// ------------------------------------------------------------------------- 
//  SRCI Robot Library                                                
// ------------------------------------------------------------------------- 
//                                                                           
//  Object:      CollisionDetectionFB                                       
//  Author:      Thorsten Brach                                                
//  Date:        2024-06-01
//
//  Description:                                              
//   
//                                                                           
//  Copyright: 
//    (C) 2024 Thorsten Brach. All rights reserved                                                                         
//                                                                           
//  Disclaimer:                                                                           
//    This project is provided without any guarantee and can be used for   
//    private and commercial purposes. Any commercial use is at the user’s 
//    own risk and responsibility.
//
// -------------------------------------------------------------------------
VAR_INPUT
  /// Start of the command at the rising edge
  Execute            : BOOL;
  /// Processing mode
  ProcessingMode     : ProcessingMode;
  ///  Defines the robot behavior after detecting the collision (at least one option must be supported):
  ReactionMode       : CollisionReactionMode;
  /// Set TRUE to activate and FALSE to deactivate "CollisionDetection".
  /// Default: TRUE
  ActivateMonitoring : BOOL;
  /// Defines the type of threshold setting (at least one option must be supported)
  ThresholdMode      : ThresholdMode;
  /// Defines the level of sensitivity of all axes.
  /// • 0..99: Sensitivity lower than robot vendor default. 
  ///          At minimum value "0" there is no sensitivity. The lower the value, the lower the sensitivity at the collision detection.
  /// • 100 (default): The value is aligned with the robot vendor-specific default value.
  /// • 101..200: Sensitivity higher than robot vendor default. At maximum value "200" highest possible sensitivity at the collision detection.
  Sensitivity        : REAL;
  /// Defines the level of sensitivity of the respective axis.
  /// Values:
  /// • 0..99: Sensitivity lower than robot vendor default. At minimum value "0" there is no sensitivity and collision detection for the respective axis. 
  ///          The lower the value, the lower the sensitivity at the collision detection.
  /// • 100 (default): The value is aligned with the robot vendor-specific default value.
  /// • 101..200: Sensitivity higher than robot vendor default. At maximum value "200" highest possible sensitivity at the collision detection.
  /// Index:
  /// • [0]: J1 First joint of the robot.
  /// • [1]: J2 Second joint of the robot.
  /// • [2] J3 Third joint of the robot.
  /// • [3] J4 Forth joint of the robot.
  /// • [4] J5 Fifth joint of the robot.
  /// • [5] J6 Six joint of the robot.
  /// • [6] J7 Seventh joint of the robot, if willbe used.
  SensitivityAxis    : ARRAY[0..6] OF REAL;
  /// Relates to "ThresholdMode" Manual. Defines the threshold of the torque for each robot axis. If the threshold is exceeded, the RA stops.
  /// Index:
  /// • [0] J1 First joint of the robot.
  /// • [1] J2 Second joint of the robot.
  /// • [2] J3 Third joint of the robot.
  /// • [3] J4 Forth joint of the robot.
  /// • [4] J5 Fifth joint of the robot.
  /// • [5] J6 Six joint of the robot.
  /// • [6] J7 Seventh joint of the robot, if will be used
  LimitAxis          : ARRAY[0..6] OF REAL;
  /// Relates to "LimitAxis". Defines the unit of the threshold.
  /// • [0]: Percentage (%) (default) O
  /// • [1]: Newton meter (Nm). O
  /// • [2] Milliampere (mA).
  UnitLimitAxis      : USINT;
  /// Defines the target sequence in which the command will be executed
  SequenceFlag       : SequenceFlag;
END_VAR
VAR_OUTPUT
  /// The command has been completed successfully
  Done               : BOOL;
  /// FB is being processed
  Busy               : BOOL;
  /// Command is transferred and confirmed by the RC
  CommandBuffered    : BOOL;
  /// The command was aborted by another command.
  CommandAborted     : BOOL;
  /// TRUE, while command is interrupted during execution and can be continued
  CommandInterrupted : BOOL;  
END_VAR

                  
                

METHOD PROTECTED OnCall
VAR_IN_OUT
  /// Robot assignment of function
  AxesGroup         : AxesGroup; 
END_VAR
                        
                      
END_METHOD
END_FUNCTION_BLOCK

/// Reads and writes specific configuration parameters on RC that are required for the RI to work
FUNCTION_BLOCK ExchangeConfigurationFB EXTENDS RobotLibraryBaseFB
// ------------------------------------------------------------------------- 
//  SRCI Robot Library                                                
// ------------------------------------------------------------------------- 
//                                                                           
//  Object:      ExchangeConfigurationFB                                       
//  Author:      Thorsten Brach                                                
//  Date:        2024-06-01
//
//  Description:                                              
//   
//                                                                           
//  Copyright: 
//    (C) 2024 Thorsten Brach. All rights reserved                                                                         
//                                                                           
//  Disclaimer:                                                                           
//    This project is provided without any guarantee and can be used for   
//    private and commercial purposes. Any commercial use is at the user’s 
//    own risk and responsibility.
//
// -------------------------------------------------------------------------

                  
                

METHOD PROTECTED OnCall
VAR_IN_OUT
  /// Robot assignment of function
  AxesGroup         : AxesGroup; 
END_VAR
                        
                      
END_METHOD
END_FUNCTION_BLOCK

/// Move the robot axes by hand
FUNCTION_BLOCK FreeDriveFB EXTENDS RobotLibraryBaseFB
// ------------------------------------------------------------------------- 
//  SRCI Robot Library                                                
// ------------------------------------------------------------------------- 
//                                                                           
//  Object:      FreeDriveFB                                       
//  Author:      Thorsten Brach                                                
//  Date:        2024-06-01
//
//  Description:                                              
//   
//                                                                           
//  Copyright: 
//    (C) 2024 Thorsten Brach. All rights reserved                                                                         
//                                                                           
//  Disclaimer:                                                                           
//    This project is provided without any guarantee and can be used for   
//    private and commercial purposes. Any commercial use is at the user’s 
//    own risk and responsibility.
//
// -------------------------------------------------------------------------
VAR_INPUT
  /// Set TRUE to change RA power state to "Enabled"
  Enable            : BOOL;
END_VAR

VAR_OUTPUT
  /// FB is being processed
  Busy              : BOOL;
  /// Command is transferred and confirmed by the RC
  CommandBuffered   : BOOL;
  /// TRUE while "FreeDrive" is active.
  Enabled           : BOOL;
  /// Receiving of input parameter values has been acknowledged by RC
  ParameterAccepted : BOOL;
END_VAR

                  
                

METHOD PROTECTED OnCall
VAR_IN_OUT
  /// Robot assignment of function
  AxesGroup         : AxesGroup; 
END_VAR
                        
                      
END_METHOD
END_FUNCTION_BLOCK

